Fanuc KAREL source: libind_mth.kl

-- Software License Agreement (BSD License)
--
-- Copyright (c) 2012, TU Delft Robotics Institute
-- All rights reserved.
--
-- Redistribution and use in source and binary forms, with or without
-- modification, are permitted provided that the following conditions
-- are met:
--
--  * Redistributions of source code must retain the above copyright
--    notice, this list of conditions and the following disclaimer.
--  * Redistributions in binary form must reproduce the above
--    copyright notice, this list of conditions and the following
--    disclaimer in the documentation and/or other materials provided
--    with the distribution.
--  * Neither the name of the TU Delft Robotics Institute nor the names
--    of its contributors may be used to endorse or promote products
--    derived from this software without specific prior written
--    permission.
--
-- THIS SOFTWARE IS PROVIDED BY THE COPYRIGHT HOLDERS AND CONTRIBUTORS
-- "AS IS" AND ANY EXPRESS OR IMPLIED WARRANTIES, INCLUDING, BUT NOT
-- LIMITED TO, THE IMPLIED WARRANTIES OF MERCHANTABILITY AND FITNESS
-- FOR A PARTICULAR PURPOSE ARE DISCLAIMED. IN NO EVENT SHALL THE
-- COPYRIGHT OWNER OR CONTRIBUTORS BE LIABLE FOR ANY DIRECT, INDIRECT,
-- INCIDENTAL, SPECIAL, EXEMPLARY, OR CONSEQUENTIAL DAMAGES (INCLUDING,
-- BUT NOT LIMITED TO, PROCUREMENT OF SUBSTITUTE GOODS OR SERVICES;
-- LOSS OF USE, DATA, OR PROFITS; OR BUSINESS INTERRUPTION) HOWEVER
-- CAUSED AND ON ANY THEORY OF LIABILITY, WHETHER IN CONTRACT, STRICT
-- LIABILITY, OR TORT (INCLUDING NEGLIGENCE OR OTHERWISE) ARISING IN
-- ANY WAY OUT OF THE USE OF THIS SOFTWARE, EVEN IF ADVISED OF THE
-- POSSIBILITY OF SUCH DAMAGE.


PROGRAM libind_mth
--------------------------------------------------------------------------------
--
-- Shared math functionality
--
-- author: G.A. vd. Hoorn
--
--------------------------------------------------------------------------------
%NOLOCKGROUP
%NOPAUSE= COMMAND + TPENABLE + ERROR
%COMMENT = 'r1'




--------------------------------------------------------------------------------
--
-- local types & constants
--
--------------------------------------------------------------------------------
const
	M_PI       =  3.14159265359
	M_1_PI     =  0.31830988618
	M_1RAD_DEG = 57.29577951318
	M_1DEG_RAD =  0.01745329252




--------------------------------------------------------------------------------
--
-- local routine prototypes
--
--------------------------------------------------------------------------------
%INCLUDE libind_mth_h




--------------------------------------------------------------------------------
--
-- Empty body
--
--------------------------------------------------------------------------------
BEGIN
END libind_mth




ROUTINE deg_to_rad
BEGIN
	RETURN (r_deg * M_1DEG_RAD)
END deg_to_rad




ROUTINE rad_to_deg
BEGIN
	RETURN (r_rad * M_1RAD_DEG)
END rad_to_deg




ROUTINE arr_deg2rad
VAR
	len_ : INTEGER
	d_   : INTEGER
BEGIN
	len_ = ARRAY_LEN(a)
	FOR d_ = 1 TO len_ DO
		a[d_] = deg_to_rad(a[d_])
	ENDFOR
END arr_deg2rad




ROUTINE arr_rad2deg
VAR
	len_ : INTEGER
	d_   : INTEGER
BEGIN
	len_ = ARRAY_LEN(a)
	FOR d_ = 1 TO len_ DO
		a[d_] = rad_to_deg(a[d_])
	ENDFOR
END arr_rad2deg
